// TIA Portal V20 export
DATA_BLOCK "DB - Equipment"   // DB4
{ S7_Optimized_Access := 'TRUE' }
// stored: MemoryReserve 100
   VAR
      TableCheckProcess1 : "UDT-TableCheck";
      TableCheckProcess2 : "UDT-TableCheck";
      "SabLaodProcess1-L" { S7_SetPoint := 'True'} : "UDT-SABload";
      "SabLaodProcess1-R" { S7_SetPoint := 'True'} : "UDT-SABload";
      "SabLaodProcess2-L" { S7_SetPoint := 'True'} : "UDT-SABload";
      "SabLaodProcess2-R" { S7_SetPoint := 'True'} : "UDT-SABload";
      Bas342 { S7_SetPoint := 'True'} : "UDT-BAS342";
   END_VAR
BEGIN
END_DATA_BLOCK
